PROGRAM main
  VAR
    HS100_PB AT %IX0.0 : BOOL := false;
    XL100_LAMP AT %QX0.0 : BOOL := false;
  END_VAR

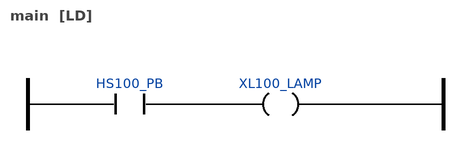
(* LD diagram, written out as Structured Text *)
XL100_LAMP := HS100_PB;
END_PROGRAM
